// TIA Portal V16 export
// export: Created 2023-01-03T15:35:08.3038254Z, ExportSetting WithDefaults, DisplayName Totally Integrated Automation Portal, DisplayVersion V16, DisplayName TIA Portal Version Control Interface, DisplayVersion V16, DisplayName TIA Portal Openness, DisplayVersion V16, DisplayName STEP 7 Professional, DisplayVersion V16, DisplayName STEP 7 Safety, DisplayVersion V16, DisplayName WinCC Advanced, DisplayVersion V16
VAR_GLOBAL   // PLC tag table "Default tag table"
   INITL_MODE AT %M3.4 : Bool;
   MNAL_MODE AT %M3.5 : Bool;
   AT_MODE AT %M3.6 : Bool;
   PTRIG1 AT %M3.7 : Bool;
   SYSTEM_ON AT %M12.0 : Bool;
   PTRIG2 AT %M12.1 : Bool;
   METAL_DETECTED AT %M12.2 : Bool;
   PTRIG3 AT %M12.3 : Bool;
   PART_SORTED AT %M12.4 : Bool;
   PLASTIC_PART_DETECTED AT %M12.5 : Bool;
   NTRIG1 AT %M12.6 : Bool;
   PLASTIC_PART_SORTED AT %M12.7 : Bool;
   Variable_Speed AT %M13.0 : Bool;
   Act_Speed_val_in_rpm AT %MW20 : Int;
   Motor_speed_monitoring_error_max AT %M13.1 : Bool;
   Motor_speed_monitoring_warning_max AT %M13.2 : Bool;
   Motor_speed_monitoring_warning_min AT %M13.3 : Bool;
   Motor_speed_monitoring_error_min AT %M13.4 : Bool;
   Motor_Overspeed_Error AT %M13.5 : Bool;
   NTRIG2 AT %M13.6 : Bool;
   SYSTEM_OFF AT %M13.7 : Bool;
   Alarms AT %MW18 : UInt;
END_VAR
